TYPE U_AXIS_STATE :
UNION

  stState             : ARRAY[1..MAX_AXIS] OF ST_AXIS_STATE;

  byState   AT %Q*    : ARRAY[1..MAX_AXIS] OF
                        ARRAY[1..SIZEOF(ST_AXIS_STATE)] OF BYTE;
END_UNION
END_TYPE

(* stored: Version 1.1.0.1, ProductVersion 3.1.4026.13
   DUT U_AXIS_STATE: Id {b336f0d2-020d-0c01-1f6f-4c95c36c4b3a} *)
